// TIA Portal V19 export
TYPE "PosFbk_Encoder_Alr"
// stored: Access Published
   STRUCT
      CommFault : Bool;   // Communication fault
      SensorFault : Bool;   // Secnsor fault
      NoRef : Bool;   // No reference (check homing)
      Resolution : Bool;   // Resolution is at 0
   END_STRUCT;
END_TYPE
